// TIA Portal V16 export
// export: Created 2022-02-04T14:40:23.591167Z, ExportSetting WithDefaults, DisplayName Totally Integrated Automation Portal, DisplayVersion V16 Update 1, DisplayName TIA Portal Version Control Interface, DisplayVersion V16, DisplayName TIA Portal Openness, DisplayVersion V16, DisplayName SINAMICS Startdrive Advanced, DisplayVersion V16 Update 5, DisplayName SINAMICS Startdrive G130, G150, S120, S150, SINAMICS MV, S210, DisplayVersion V16 Update 5, DisplayName SINAMICS Startdrive G110M, G120, G120C, G120D, G120P, G115D, DisplayVersion V16 Update 5, DisplayName STEP 7 Professional, DisplayVersion V16, DisplayName STEP 7 Safety, DisplayVersion V16, DisplayName WinCC Advanced, DisplayVersion V16, DisplayName SIMATIC Visualization Architect, DisplayVersion V16
DATA_BLOCK "FB_Rollout_Zone_DB"   // DB31
VERSION : 0.1
// stored: AutoNumber true, InstanceOfName FB_Rollout_Zone, InstanceOfType FB
"FB_Rollout_Zone"
   // VAR_INPUT
   //    lift_returning : Bool;
   //    packet_ready : Bool;
   //    m_322_sensor : Bool;
   //    m_324_sensor : Bool;
   //    m_324_sync : Bool;
   //    lift_down_sensor : Bool;
   //    lift_up_sensor : Bool;
   // END_VAR
   // VAR_OUTPUT
   //    packet_released : Bool;
   // END_VAR
   // VAR_IN_OUT
   //    rolling_packet { ExternalAccessible := 'False'; ExternalVisible := 'False'; ExternalWritable := 'False'} : Bool;
   // END_VAR
   // VAR RETAIN
   //    busyM321 : Bool;
   //    busyM322 : Bool;
   //    busyM322_old : Bool;
   //    busyM324 : Bool;
   //    m_324_ready : Bool;
   //    m_324_move_trig : Bool;
   //    m_324_sens_old : Bool;
   //    m_324_sync_old : Bool;
   //    safe_rollout_timer : TON;
   //    delay_start_m_324 { S7_SetPoint := 'True'} : TON;
   //    busy321_timer { S7_SetPoint := 'True'} : TON;
   //    busy322_timer { S7_SetPoint := 'True'} : TOF;
   //    busy324_timer { S7_SetPoint := 'True'} : TOF;
   // END_VAR
BEGIN
END_DATA_BLOCK
